Universal Robots PolyScope program: shaft_turning_touch_only.urp

Program shaft_turning_touch_only (installation=default directory=/programs/wrs2020 createdIn=5.7.0.90932 lastSavedIn=5.7.0.90932 robotSerialNumber=20205500607)
Calibrated DH parameters: a=[0.000096, -0.337, -0.383372, 0.000118, 0.000015, 0]; d=[0.162724, 79.377998, -95.545185, 16.300583, 0.099689, 0.099499]; alpha=[1.569249, 0.003272, 0.005201, 1.570041, -1.570219, 0]; deltaTheta=[0, 0.65664, 5.410619, 0.215927, -0.000001, 0]
Robot Program (runOnlyOnce=false)
  URCap Gripper (Robotiq_Grippers, Robotiq Inc.) dataModel(position=0.0, force=100.0, speed=100.0, positionInDouble=0.0, forceInDouble=100.0, speedInDouble=100.0, slaveIds=[9], blocking=true)
  SuppressedNode
    Wait Sleep waitTime=0.5
  MoveL speed 1000 mm/s, acceleration 1500 mm/s^2 (useActiveTCP=true) feature=Base
    Waypoint at_shaft: TCP in base x=292.462 y=-172.285 z=28.427 mm, rx=-0.0168 ry=3.1097 rz=0.0286 rad; joints [124.781, -97.407, 145.354, -138.076, -87.656, 34.218] deg; TCP offset x=0 y=0 z=165 mm, rx=0 ry=0 rz=0 rad
  SuppressedNode
    Popup Message (haltProgram=false message=ok to turn shaft inputType=Text)
  SuppressedNode
    MoveJ speed 60 deg/s, acceleration 80 deg/s^2 (useActiveTCP=false) tcp=gripper_85_tip; feature=Base
      Waypoint above: TCP in base x=292.462 y=-172.285 z=62.712 mm, rx=-0.0168 ry=3.1097 rz=0.0286 rad; joints [124.809, -102.836, 142.411, -129.703, -87.649, 34.201] deg
  MoveL speed 800 mm/s, acceleration 1200 mm/s^2 (useActiveTCP=true) feature=Base
    Waypoint at_shaft_left: TCP in base x=327.5 y=-167.988 z=30.411 mm, rx=-0.0193 ry=2.7762 rz=0.0232 rad; joints [116.268, -99.201, 153.713, -153.118, -70.614, 27.035] deg
    Waypoint up (Relative): motionParameters(blendRadius=0); relativeFromPosition TCP in base x=328.863 y=-168.012 z=30.45 mm, rx=-0.0193 ry=2.7762 rz=0.0231 rad; joints [116.536, -98.949, 153.569, -153.324, -70.655, 27.315] deg; TCP in base x=328.811 y=-168.489 z=49.894 mm, rx=-0.0193 ry=2.7764 rz=0.0234 rad; joints [116.504, -103.393, 151.919, -147.191, -70.642, 27.246] deg
    SuppressedNode
      Waypoint at_right_up: motionParameters(blendRadius=0); TCP in base x=326.174 y=-168.134 z=45.287 mm, rx=-0.0194 ry=2.7762 rz=0.0231 rad; joints [116.005, -102.956, 152.62, -148.176, -70.566, 26.73] deg
    SuppressedNode
      Waypoint at_right: motionParameters(blendRadius=0); TCP in base x=293.492 y=-172.285 z=29.381 mm, rx=0.0082 ry=-2.6779 rz=-0.0282 rad; joints [139.588, -81.714, 127.322, -114.069, -105.719, 52.27] deg
    Waypoint at_shaft: TCP in base x=292.462 y=-172.285 z=28.427 mm, rx=-0.0168 ry=3.1097 rz=0.0286 rad; joints [124.781, -97.407, 145.354, -138.076, -87.656, 34.218] deg
